{attribute 'GeneratedUsingTerminal: EL6201-0000-0017'}
{attribute addProperty BoxType "EL6201-0000-0017"}
{attribute addProperty Id "Slave_7A_DO0BOOL1Slave_7A_DO1BOOL1Slave_7A_DO2BOOL1Slave_7A_DO3BOOL1Slave_7B_DO0BOOL1Slave_7B_DO1BOOL1Slave_7B_DO2BOOL1Slave_7B_DO3BOOL1"}
{attribute addProperty CRC "1477708597"}
{attribute addProperty Size "8"}
TYPE Slave_7_Outputs_58140B35 :
STRUCT
	{attribute addProperty Name "Slave_7A_DO0"}
	Slave_7A_DO0 : BOOL;
	{attribute addProperty Name "Slave_7A_DO1"}
	Slave_7A_DO1 : BOOL;
	{attribute addProperty Name "Slave_7A_DO2"}
	Slave_7A_DO2 : BOOL;
	{attribute addProperty Name "Slave_7A_DO3"}
	Slave_7A_DO3 : BOOL;
	{attribute addProperty Name "Slave_7B_DO0"}
	Slave_7B_DO0 : BOOL;
	{attribute addProperty Name "Slave_7B_DO1"}
	Slave_7B_DO1 : BOOL;
	{attribute addProperty Name "Slave_7B_DO2"}
	Slave_7B_DO2 : BOOL;
	{attribute addProperty Name "Slave_7B_DO3"}
	Slave_7B_DO3 : BOOL;
END_STRUCT
END_TYPE

(* stored: Version 1.2.0.0, ProductVersion 3.1.4024.9
   DUT Slave_7_Outputs_58140B35: Id {dc8dd4e6-a261-4953-b411-2484879a3390} *)
